(* PLC project MethodMemberFixture *)

FUNCTION_BLOCK FB_TEST

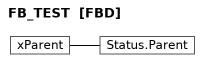
(* FBD diagram, written out as Structured Text *)
Status.Parent := xParent;

METHOD Compute
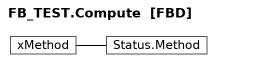
(* FBD diagram, written out as Structured Text *)
Status.Method := xMethod;
END_METHOD
END_FUNCTION_BLOCK
